{attribute 'GeneratedUsingTerminal: ER7041-0002-0024'}
{attribute addProperty BoxType "ER7041-0002-0024"}
{attribute addProperty Id "Ready_to_enableBOOL1ReadyBOOL1WarningBOOL1ErrorBOOL1Moving_positiveBOOL1Moving_negativeBOOL1Torque_reducedBOOL1Digital_input_1BOOL1Digital_input_2BOOL1Sync_errorBOOL1TxPDO_ToggleBOOL1"}
{attribute addProperty CRC "3061405765"}
{attribute addProperty Size "11"}
TYPE Status_B6795845 :
STRUCT
	{attribute addProperty Name "Ready_to_enable"}
	Ready_to_enable : BOOL;
	{attribute addProperty Name "Ready"}
	Ready : BOOL;
	{attribute addProperty Name "Warning"}
	Warning : BOOL;
	{attribute addProperty Name "Error"}
	Error : BOOL;
	{attribute addProperty Name "Moving_positive"}
	Moving_positive : BOOL;
	{attribute addProperty Name "Moving_negative"}
	Moving_negative : BOOL;
	{attribute addProperty Name "Torque_reduced"}
	Torque_reduced : BOOL;
	{attribute addProperty Name "Digital_input_1"}
	Digital_input_1 : BOOL;
	{attribute addProperty Name "Digital_input_2"}
	Digital_input_2 : BOOL;
	{attribute addProperty Name "Sync_error"}
	Sync_error : BOOL;
	{attribute addProperty Name "TxPDO_Toggle"}
	TxPDO_Toggle : BOOL;
END_STRUCT
END_TYPE

(* stored: Version 1.2.0.0, ProductVersion 3.1.4024.9
   DUT Status_B6795845: Id {c8796fa2-46b2-4e33-a6b2-aa8a51fb361e} *)
